{region '#Template'}
	{attribute 'Version' := '5.0.0.0'}
	{attribute 'Tags' := '"LCID": "1031", "Text": "Universal, Control, Hysteresis"'}
	{attribute 'Tags' := '"LCID": "1033", "Text": "Universal, Control, Hysteresis"'}
	{attribute 'Using' := '"Type": "Template", "URI": "EC_ID"'}
	{attribute 'Using' := '"Type": "Template", "URI": "BA2_Param"'}
	{attribute 'Description' := '"LCID": "1031", "Text": "Hysterese"'}
	{attribute 'Description' := '"LCID": "1033", "Text": "Hysteresis"'}
{endregion}
FUNCTION_BLOCK FB_BA_Hys_21 EXTENDS FB_BA_View
VAR_INPUT
	bEn 					: BOOL := TRUE;	
	fIn						: REAL;
END_VAR
VAR_OUTPUT
	bDst					: BOOL;
END_VAR
VAR_INPUT CONSTANT
	HysPreAlarmOn			: FB_BA_AV_Op;		
	HysPreAlarmOff			: FB_BA_AV_Op;		
	HysMainAlarmOn			: FB_BA_AV_Op;		
	HysMainAlarmOff			: FB_BA_AV_Op;	
	DstPreAlarm				: FB_BA_BV;
	DstMainAlarm			: FB_BA_BV;
END_VAR
VAR
	HysPreAlarm				: FB_BA_Swi2P;
	HysMainAlarm			: FB_BA_Swi2P;
END_VAR

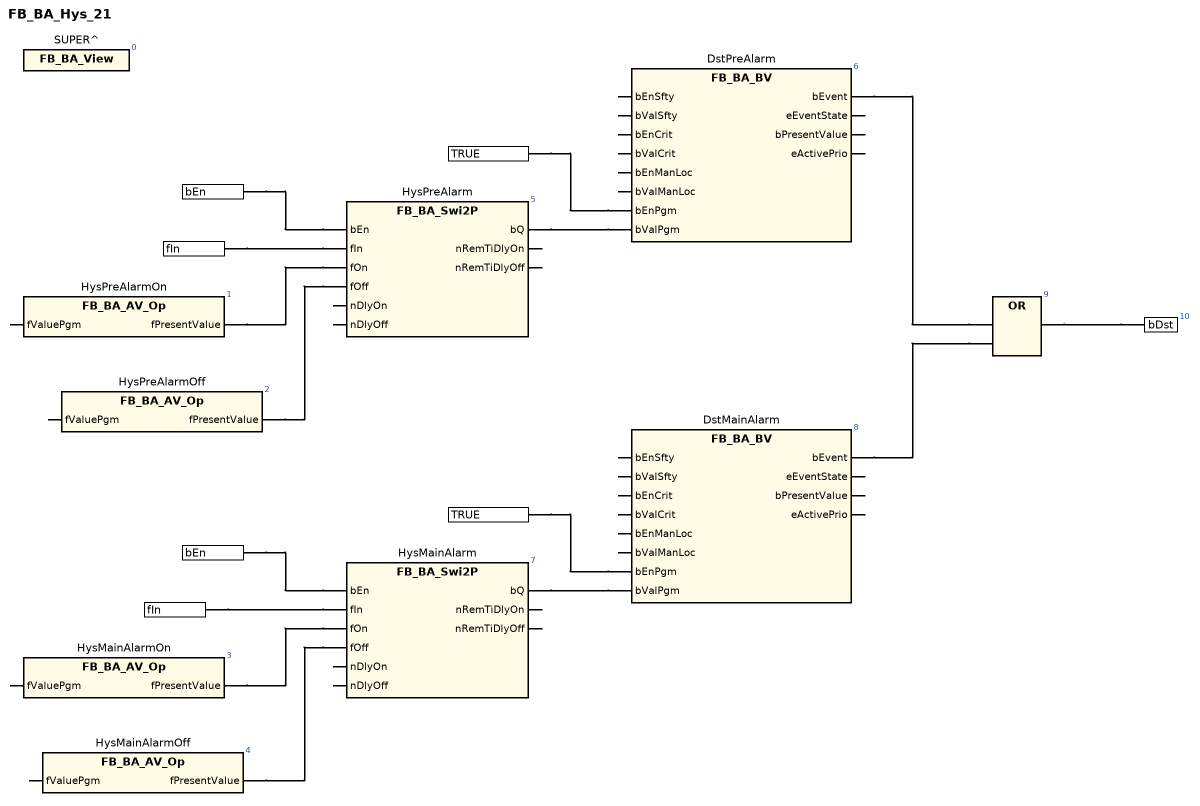
SUPER^(); // FB_BA_View
HysPreAlarmOn(); // FB_BA_AV_Op
HysPreAlarmOff(); // FB_BA_AV_Op
HysMainAlarmOn(); // FB_BA_AV_Op
HysMainAlarmOff(); // FB_BA_AV_Op
HysPreAlarm(bEn := bEn, fIn := fIn, fOn := HysPreAlarmOn.fPresentValue, fOff := HysPreAlarmOff.fPresentValue); // FB_BA_Swi2P
DstPreAlarm(bEnPgm := TRUE, bValPgm := HysPreAlarm.bQ); // FB_BA_BV
HysMainAlarm(
    bEn := bEn,
    fIn := fIn,
    fOn := HysMainAlarmOn.fPresentValue,
    fOff := HysMainAlarmOff.fPresentValue); // FB_BA_Swi2P
DstMainAlarm(bEnPgm := TRUE, bValPgm := HysMainAlarm.bQ); // FB_BA_BV
bDst := DstPreAlarm.bEvent OR DstMainAlarm.bEvent;

METHOD FB_init : BOOL
VAR_INPUT
	bInitRetains : BOOL; // if TRUE, the retain variables are initialized (warm start / cold start)
	bInCopyCode : BOOL;  // if TRUE, the instance afterwards gets moved into the copy code (online change)
END_VAR
HysPreAlarmOn.iParent						:= THIS^;  
HysPreAlarmOn.iLabel						:= LblCtl_PreAlarmLimitMAX;    	
HysPreAlarmOn.eUnit							:= E_BA_Unit.ePressure_Pascals;							 	 
HysPreAlarmOn.fValueRm						:= 200;			
HysPreAlarmOn.fCOVIncrement					:= BA2_Param.fDefCOVIncrement;		

HysPreAlarmOff.iParent						:= THIS^;
HysPreAlarmOff.iLabel						:= LblCtl_PreAlarmLimitMIN;    	
HysPreAlarmOff.eUnit						:= E_BA_Unit.ePressure_Pascals;							 	 
HysPreAlarmOff.fValueRm						:= 150;			
HysPreAlarmOff.fCOVIncrement				:= BA2_Param.fDefCOVIncrement;		
							
HysMainAlarmOn.iParent						:= THIS^;
HysMainAlarmOn.iLabel						:= LblCtl_MainAlarmLimitMAX;    										 	 
HysMainAlarmOn.eUnit						:= E_BA_Unit.ePressure_Pascals;
HysMainAlarmOn.fValueRm						:= 350;			
HysMainAlarmOn.fCOVIncrement				:= BA2_Param.fDefCOVIncrement;		
							
HysMainAlarmOff.iParent						:= THIS^;
HysMainAlarmOff.iLabel						:= LblCtl_MainAlarmLimitMIN;   								 	 
HysMainAlarmOff.eUnit						:= E_BA_Unit.ePressure_Pascals;
HysMainAlarmOff.fValueRm					:= 300;			
HysMainAlarmOff.fCOVIncrement				:= BA2_Param.fDefCOVIncrement;		

DstPreAlarm.iParent							:= THIS^;
DstPreAlarm.iLabel							:= LblCtl_PreAlarmFault;    
DstPreAlarm.sActiveText 					:= txtEvent_Maintenace;
DstPreAlarm.sInactiveText 					:= txtEvent_Normal;
DstPreAlarm.bEnManualRm						:= FALSE;	//	Priority  8	
DstPreAlarm.bValManualRm					:= FALSE;	//	Priority  8
DstPreAlarm.nEventClassID					:= EC_ID.NC50;
DstPreAlarm.stTimeDelay.nToNormal			:= 0;
DstPreAlarm.stTimeDelay.nToAbnormal			:= 0;
DstPreAlarm.bAlarmValue						:= TRUE;
DstPreAlarm.aEventTransitionText[1]			:= txtEvent_Disturb;
DstPreAlarm.aEventTransitionText[2]			:= txtEvent_None;
DstPreAlarm.aEventTransitionText[3]			:= txtEvent_Normal;
DstPreAlarm.bEventDetectionEnable			:= TRUE;
DstPreAlarm.eEnPlantLock					:= E_BA_LockPriority.eNoLock;	

DstMainAlarm.iParent						:= THIS^;
DstMainAlarm.iLabel							:= LblCtl_MainAlarmFault;    
DstMainAlarm.sActiveText 					:= txtEvent_Triggered;
DstMainAlarm.sInactiveText 					:= txtEvent_Normal;
DstMainAlarm.bEnManualRm					:= FALSE;	//	Priority  8	
DstMainAlarm.bValManualRm					:= FALSE;	//	Priority  8
DstMainAlarm.nEventClassID					:= EC_ID.NC30;
DstMainAlarm.stTimeDelay.nToNormal			:= 0;
DstMainAlarm.stTimeDelay.nToAbnormal		:= 0;
DstMainAlarm.bAlarmValue					:= TRUE;
DstMainAlarm.aEventTransitionText[1]		:= txtEvent_Triggered;
DstMainAlarm.aEventTransitionText[2]		:= txtEvent_Error;
DstMainAlarm.aEventTransitionText[3]		:= txtEvent_Normal;
DstMainAlarm.bEventDetectionEnable			:= TRUE;
DstMainAlarm.eEnPlantLock					:= E_BA_LockPriority.eNoLock;
END_METHOD

END_FUNCTION_BLOCK

(* stored: Version 1.1.0.1, ProductVersion 3.1.4024.12
   POU FB_BA_Hys_21: Id {3f32bdd7-a204-491a-9937-7b510a5ff557}, SpecialFunc None
   Method FB_init: Id {708c9e99-f714-465f-bb1f-19e526ec0016} *)
